(* IEC 61131-3 sources: ICSML/Codesys_V3/Function Blocks/BStep_L.pou, 1 file *)

(* ---- BStep_L.pou ---- *)
(*#-#-#-#-#-#-#-#-#-#---Declaration---#-#-#-#-#-#-#-#-#-#-#-#-#*)

(*
	Binary Step Activation Layer
*)
FUNCTION_BLOCK PUBLIC BStep_L IMPLEMENTS Activation
VAR
	// Input and Output dataMem variables
	input_i: dataMem;
	output_i: dataMem;
END_VAR
(*#-#-#-#-#-#-#-#-#-#---Implementation---#-#-#-#-#-#-#-#-#-#-#-#-#*)
